FUNCTION_BLOCK fb_BusPingEvent_1
VAR_INPUT
	 I_sID         			:STRING(10);     // Geräte-ID (z.B. '12345')
	 I_sReceivedString		:STRING(255);	
	 I_iInstID				:INT := 17;						(* Instanz ID *)
	 I_bTasterMode			:BOOL;
	 I_bReset				:BOOL;
END_VAR
VAR_OUTPUT
	Q_bOut					:BOOL;
END_VAR
VAR
	findString0				:STRING ;
	findString1				:STRING ;
	findString2				:STRING ;
	findString3				:STRING ;
	findString4				:STRING ;
	
END_VAR


findString0 := CONCAT(I_sID,'.');
findString0 := CONCAT(findString0,'BTN');
findString0 := CONCAT(findString0,'.');
findString0 := CONCAT(findString0,INT_TO_STRING(I_iInstID));
findString0 := CONCAT(findString0,'.');
findString0 := CONCAT(findString0,'rSTATUS');

(* Wenn ein Taster gedrückt wird *)
findString1 := CONCAT(I_sID,'.');
findString1 := CONCAT(findString1,'BTN');
findString1 := CONCAT(findString1,'.');
findString1 := CONCAT(findString1,INT_TO_STRING(I_iInstID));
findString1 := CONCAT(findString1,'.');
findString1 := CONCAT(findString1,'STATUS');

(* Wenn Ein Temperatur Event Kommt *)
findString2 := CONCAT(I_sID,'.');
findString2 := CONCAT(findString2,'TEMP.1.STATUS');
(* Wenn Ein Feuchtigkeit Event Kommt *)
findString3 := CONCAT(I_sID,'.');
findString3 := CONCAT(findString3,'RHD.1.STATUS');
(* Wenn Ein Helligkeit Event Kommt *)
findString4 := CONCAT(I_sID,'.');
findString4 := CONCAT(findString4,'BRS.1.STATUS');

IF I_bReset
THEN
	Q_bOut := FALSE;
ELSE
	IF FIND(I_sReceivedString,findString0) >0 
		OR (FIND(I_sReceivedString,findString1) >0 
		AND I_bTasterMode)
		OR (FIND(I_sReceivedString,findString2) >0 
		AND I_bTasterMode)
		OR (FIND(I_sReceivedString,findString3) >0 
		AND I_bTasterMode)
		OR (FIND(I_sReceivedString,findString4) >0 
		AND I_bTasterMode)
		
	THEN
		Q_bOut := TRUE;
	ELSE
		Q_bOut := FALSE;
	END_IF
END_IF

END_FUNCTION_BLOCK

(* stored: Version 1.1.0.1, ProductVersion 3.1.4024.12
   POU fb_BusPingEvent_1: Id {abc99c70-09f0-4b0b-88af-b54d69408347}, SpecialFunc None *)
